TYPE ref_eje_output :
STRUCT
	out_flg_ejeVac : BOOL;
	out_flg_ejeBrk : BOOL;
END_STRUCT
END_TYPE

(* stored: Version 1.1.0.1, ProductVersion 3.1.4024.11
   DUT ref_eje_output: Id {5c1e12ea-255c-4629-914a-616589b3e4e6} *)
